Staubli VAL3: copyFile.pgx

program copyFile()
  local bool l_bRes
begin
  //copy file or folder from sFrom to sTo
  l_bRes=$copy(sFrom,sTo)
  if l_bRes
    gotoxy(1,3)
    put("拷贝文件:"+sFrom+"至"+sTo)
  else
    gotoxy(1,3)
    put("拷贝文件出错:"+sFrom)
  endIf

end
